TYPE ST_LeakTester :
STRUCT
	
	State							: E_LeakTester_State;	
	CMD								: ST_GeneralStationCMD;
	Status							: ST_StationStatus;
	
END_STRUCT
END_TYPE

(* stored: Version 1.1.0.1, ProductVersion 3.1.4024.13
   DUT ST_LeakTester: Id {9b2abc05-6e52-486d-bd5f-5eef4986d306} *)
